(* IEC 61131-3 sources: lc3-demo-project/src, 1 file *)

(* ---- program.iecst ---- *)
/*  This sample contains a program to count up or down.  */
PROGRAM Counter

	VAR
    	/* If 'up' = 'TRUE', counter counts up. */
		up : BOOL;
		/* 'count' is incremented/decremented by '3' for each cycle. */
		count : INT;
	END_VAR

	IF up THEN
		count := count + 3;
	ELSE
		count := count - 3;
	END_IF;

END_PROGRAM
